FUNCTION_BLOCK XY_VIEW (* View of a Two-Dimensional Mechanism *)
  (* Standard: IEC 61499; Classification: View; ApplicationDomain: Material Handling *)
  (* Version 0.0, 2006-06-20, JHC, Holobloc Inc, Copied/Modified from MECH_VIEW *)
  (* Compiler header: package fb.rt.mva; *)
  (* Compiler classdef: public class XY_VIEW extends XABS_VIEW *)
  (* Compiler Java Sun JDK 1.5.0 *)
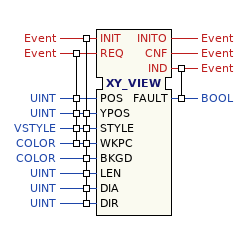
  EVENT_INPUT
    INIT WITH STYLE, WKPC, BKGD, LEN, DIA, DIR, YPOS; (* Initialize *)
    REQ WITH POS, STYLE, WKPC, YPOS; (* Update the display *)
  END_EVENT
  EVENT_OUTPUT
    INITO; (* Initialized *)
    CNF; (* Display Updated *)
    IND WITH FAULT; (* Change in FAULT status *)
  END_EVENT
  VAR_INPUT
    POS : UINT; (* X-position, {0..100}% *)
    YPOS : UINT; (* Y-position, {0..100}% *)
    STYLE : VSTYLE := RING; (* Workpiece style *)
    WKPC : COLOR := blue; (* Foreground Color *)
    BKGD : COLOR := blue; (* Background Color *)
    LEN : UINT; (* Length/Width in Diameters *)
    DIA : UINT; (* Workpiece Diameter *)
    DIR : UINT; (* Direction 0=>100%: 0=UL/LR,1=UR/LL,2=LR/UL,3=LL/UR *)
  END_VAR
  VAR_OUTPUT
    FAULT : BOOL; (* 0=Normal,1=Fault *)
  END_VAR
END_FUNCTION_BLOCK
